// TIA Portal V19 export
DATA_BLOCK "INTERLOCK DB"   // DB38
{ S7_Optimized_Access := 'FALSE' }
   VAR RETAIN
      ERROR : Bool;
      "CIT-101 HH" : Real;
      "PS-201 COIL" : Bool;
      "DPT-101 pressure is higher" : Real;
      "DPT-201" : Real;
      "UF INTERLOCK FOR LT-102 AND LT201 SYSTER PAUSE BUFF" : Int;
      "PT-601 HH SET" : Real;
      "pHIT-601 HIGH" : Real;
      "pHIT-601 LOW" : Real;
      "RIT-601 HIGH" : Real;
      "RIT-601 LOW" : Real;
      "UV ONLY ALARM" : Real;
      BUFF : Struct
         "PS-101 BUFF" : Int;
         "CIT-101 HH BUFF" : Int;
         "PS-201 BUFF" : Int;
         "DPT-101 pressure is higher" : Int;
         "DPT-201" : Int;
         "PT-601 HH BUFF" : Int;
         "pHIT-601 HIGH/LOW" : Int;
         "RIT-601 HIGH BUFF" : Int;
         "UV ONLY ALARM" : Bool;
      END_STRUCT;
      "TIMER SET" : Struct
         "CIT-101 HH TIMER SET" : Int;
         "RIT-601 HIGH TIMER SET" : Int;
      END_STRUCT;
      "TIMER PV" : Struct
         "CIT-101 HH TIMER PV" : Int;
         "RIT-601 HIGH TIMER PV" : Int;
      END_STRUCT;
   END_VAR
BEGIN
END_DATA_BLOCK
